//Converts a RobotPoseSimple 2 RobotPose, assuming an error of 0
//NOTE: the reverse conversion is not needed because of polymorphmism of RobotPose, see Defintion of RobotPose STRUCT
FUNCTION RPS2RP : RobotPose
VAR_INPUT
	pose: RobotPose;
END_VAR
VAR
END_VAR

RPS2RP.x   		:= pose.x;
RPS2RP.y		:= pose.y;
RPS2RP.theta  	:= pose.theta;
RPS2RP.e		:= 0;

END_FUNCTION

(* stored: Version 1.1.0.1, ProductVersion 3.1.4024.11
   POU RP2RPS: Id {32517886-ccfa-45ed-a75b-c9097123353f}, SpecialFunc None *)
